// TIA Portal V20 export
DATA_BLOCK "LER_Recipe_DB"   // DB116
// stored: Access Published, InstanceOfName LER_Recipe, InstanceOfType FB
"LER_Recipe"
   // VAR_INPUT
   //    enable : Bool;
   //    applyBT : Bool;
   // END_VAR
   // VAR_IN_OUT
   //    parameterRecipeInterface : "HMI_IF_Parameter_LIstRecipe_Interface";
   //    parameterListSV : "HMI_IF_Parameter_ListRecipe_UDT";
   //    parameterListPV : "HMI_IF_Parameter_ListRecipe_UDT";
   // END_VAR
BEGIN
END_DATA_BLOCK
